Staubli VAL3: io.pjx

--- io.pjx ---
Parameters version=s7.2 stackSize=0 millimeterUnit=true
Data file=io.dtx

--- io.dtx ---
public aio CBT_TEMP = {link=CBT_TEMP}
public aio CPU_TEMP = {link=CPU_TEMP}
public aio MbAI_a8Axispose = {link=MbAI_a8Axispose}
public aio MbAI_aCurPosH = {link=MbAI_aCurPosH}
public aio MbAI_aCurPosL = {link=MbAI_aCurPosL}
public aio MbAI_aUnused4 = {link=MbAI_aUnused4}
public aio MbAI_b8MotorErr = {link=MbAI_b8MotorErr}
public aio MbAI_b8MotorPow = {link=MbAI_b8MotorPow}
public aio MbAI_bAxis7Reac = {link=MbAI_bAxis7Reac}
public aio MbAI_bAxis8Reac = {link=MbAI_bAxis8Reac}
public aio MbAI_bBackHome = {link=MbAI_bBackHome}
public aio MbAI_bDownLimit = {link=MbAI_bDownLimit}
public aio MbAI_bEndCycl = {link=MbAI_bEndCycl}
public aio MbAI_bHomeDone = {link=MbAI_bHomeDone}
public aio MbAI_bHomeLimit = {link=MbAI_bHomeLimit}
public aio MbAI_bIsHome = {link=MbAI_bIsHome}
public aio MbAI_bMotorErro = {link=MbAI_bMotorErro}
public aio MbAI_bMotorPowe = {link=MbAI_bMotorPowe}
public aio MbAI_bOutAlarm = {link=MbAI_bOutAlarm}
public aio MbAI_bPowerOn = {link=MbAI_bPowerOn}
public aio MbAI_bStartCycl = {link=MbAI_bStartCycl}
public aio MbAI_bUnused1 = {link=MbAI_bUnused1}
public aio MbAI_bUnused10 = {link=MbAI_bUnused10}
public aio MbAI_bUnused11 = {link=MbAI_bUnused11}
public aio MbAI_bUnused2 = {link=MbAI_bUnused2}
public aio MbAI_bUnused3 = {link=MbAI_bUnused3}
public aio MbAI_bUnused5 = {link=MbAI_bUnused5}
public aio MbAI_bUnused6 = {link=MbAI_bUnused6}
public aio MbAI_bUnused7 = {link=MbAI_bUnused7}
public aio MbAI_bUnused8 = {link=MbAI_bUnused8}
public aio MbAI_bUnused9 = {link=MbAI_bUnused9}
public aio MbAI_bUpLimit = {link=MbAI_bUpLimit}
public aio MbAO_aAxis7Puls = {link=MbAO_aAxis7Puls}
public aio MbAO_aAxis8Puls = {link=MbAO_aAxis8Puls}
public aio MbAO_aJogVelo = {link=MbAO_aJogVelo}
public aio MbAO_aJogVelo8 = {link=MbAO_aJogVelo8}
public aio MbAO_aMoveDis = {link=MbAO_aMoveDis}
public aio MbAO_aMoveDis8 = {link=MbAO_aMoveDis8}
public aio MbAO_aMovePosH = {link=MbAO_aMovePosH}
public aio MbAO_aMovePosH8 = {link=MbAO_aMovePosH8}
public aio MbAO_aMovePosL = {link=MbAO_aMovePosL}
public aio MbAO_aMovePosL8 = {link=MbAO_aMovePosL8}
public aio MbAO_aUnused10 = {link=MbAO_aUnused10}
public aio MbAO_aUnused11 = {link=MbAO_aUnused11}
public aio MbAO_aUnused6 = {link=MbAO_aUnused6}
public aio MbAO_aUnused7 = {link=MbAO_aUnused7}
public aio MbAO_aUnused8 = {link=MbAO_aUnused8}
public aio MbAO_aUnused9 = {link=MbAO_aUnused9}
public aio MbAO_aVelocity = {link=MbAO_aVelocity}
public aio MbAO_aVelocity8 = {link=MbAO_aVelocity8}
public aio MbAO_b7Axis = {link=MbAO_b7Axis}
public aio MbAO_b8Axis = {link=MbAO_b8Axis}
public aio MbAO_bAxis7Dire = {link=MbAO_bAxis7Dire}
public aio MbAO_bAxis7Home = {link=MbAO_bAxis7Home}
public aio MbAO_bAxis8Dire = {link=MbAO_bAxis8Dire}
public aio MbAO_bMoveDir = {link=MbAO_bMoveDir}
public aio MbAO_bMoveDirM = {link=MbAO_bMoveDirM}
public aio MbAO_bMovePos8 = {link=MbAO_bMovePos8}
public aio MbAO_bMoveToPos = {link=MbAO_bMoveToPos}
public aio MbAO_bRecordPos = {link=MbAO_bRecordPos}
public aio MbAO_bResetErr = {link=MbAO_bResetErr}
public aio MbAO_bStopMotor = {link=MbAO_bStopMotor}
public aio MbAO_bUnused1 = {link=MbAO_bUnused1}
public aio MbAO_bUnused2 = {link=MbAO_bUnused2}
public aio MbAO_bUnused3 = {link=MbAO_bUnused3}
public aio MbAO_bUnused4 = {link=MbAO_bUnused4}
public aio MbAO_bUnused5 = {link=MbAO_bUnused5}
public aio cCounts = {link=cCounts}
public aio cCurrPos = {link=cCurrPos}
public aio cLatchPos = {link=cLatchPos}
public aio cPrstPos = {link=cPrstPos}
public dio CASTING = {link=CASTING}
public dio DSI_BOARD = {link=DSI_BOARD}
public dio GLOBAL_PTC = {link=GLOBAL_PTC}
public dio MOTOR_1_3_5 = {link=MOTOR_1_3_5}
public dio MOTOR_2_4_6 = {link=MOTOR_2_4_6}
public dio SECTEUR_OK = {link=SECTEUR_OK}
public dio b2In0 = {link=BasicIO-2\%I0}
public dio b2In1 = {link=BasicIO-2\%I1}
public dio b2In10 = {link=BasicIO-2\%I10}
public dio b2In11 = {link=BasicIO-2\%I11}
public dio b2In12 = {link=BasicIO-2\%I12}
public dio b2In13 = {link=BasicIO-2\%I13}
public dio b2In14 = {link=BasicIO-2\%I14}
public dio b2In15 = {link=BasicIO-2\%I15}
public dio b2In2 = {link=BasicIO-2\%I2}
public dio b2In3 = {link=BasicIO-2\%I3}
public dio b2In4 = {link=BasicIO-2\%I4}
public dio b2In5 = {link=BasicIO-2\%I5}
public dio b2In6 = {link=BasicIO-2\%I6}
public dio b2In7 = {link=BasicIO-2\%I7}
public dio b2In8 = {link=BasicIO-2\%I8}
public dio b2In9 = {link=BasicIO-2\%I9}
public dio b2Out0 = {link=BasicIO-2\%Q0}
public dio b2Out1 = {link=BasicIO-2\%Q1}
public dio b2Out10 = {link=BasicIO-2\%Q10}
public dio b2Out11 = {link=BasicIO-2\%Q11}
public dio b2Out12 = {link=BasicIO-2\%Q12}
public dio b2Out13 = {link=BasicIO-2\%Q13}
public dio b2Out14 = {link=BasicIO-2\%Q14}
public dio b2Out15 = {link=BasicIO-2\%Q15}
public dio b2Out2 = {link=BasicIO-2\%Q2}
public dio b2Out3 = {link=BasicIO-2\%Q3}
public dio b2Out4 = {link=BasicIO-2\%Q4}
public dio b2Out5 = {link=BasicIO-2\%Q5}
public dio b2Out6 = {link=BasicIO-2\%Q6}
public dio b2Out7 = {link=BasicIO-2\%Q7}
public dio b2Out8 = {link=BasicIO-2\%Q8}
public dio b2Out9 = {link=BasicIO-2\%Q9}
public dio bIn0 = {link=BasicIO-1\%I0}
public dio bIn1 = {link=BasicIO-1\%I1}
public dio bIn10 = {link=BasicIO-1\%I10}
public dio bIn11 = {link=BasicIO-1\%I11}
public dio bIn12 = {link=BasicIO-1\%I12}
public dio bIn13 = {link=BasicIO-1\%I13}
public dio bIn14 = {link=BasicIO-1\%I14}
public dio bIn15 = {link=BasicIO-1\%I15}
public dio bIn2 = {link=BasicIO-1\%I2}
public dio bIn3 = {link=BasicIO-1\%I3}
public dio bIn4 = {link=BasicIO-1\%I4}
public dio bIn5 = {link=BasicIO-1\%I5}
public dio bIn6 = {link=BasicIO-1\%I6}
public dio bIn7 = {link=BasicIO-1\%I7}
public dio bIn8 = {link=BasicIO-1\%I8}
public dio bIn9 = {link=BasicIO-1\%I9}
public dio bOut0 = {link=BasicIO-1\%Q0}
public dio bOut1 = {link=BasicIO-1\%Q1}
public dio bOut10 = {link=BasicIO-1\%Q10}
public dio bOut11 = {link=BasicIO-1\%Q11}
public dio bOut12 = {link=BasicIO-1\%Q12}
public dio bOut13 = {link=BasicIO-1\%Q13}
public dio bOut14 = {link=BasicIO-1\%Q14}
public dio bOut15 = {link=BasicIO-1\%Q15}
public dio bOut2 = {link=BasicIO-1\%Q2}
public dio bOut3 = {link=BasicIO-1\%Q3}
public dio bOut4 = {link=BasicIO-1\%Q4}
public dio bOut5 = {link=BasicIO-1\%Q5}
public dio bOut6 = {link=BasicIO-1\%Q6}
public dio bOut7 = {link=BasicIO-1\%Q7}
public dio bOut8 = {link=BasicIO-1\%Q8}
public dio bOut9 = {link=BasicIO-1\%Q9}
public dio cEnLatch = {link=cEnLatch}
public dio cEnPrst = {link=cEnPrst}
public dio cHwErr = {link=cHwErr}
public dio cLatch = {link=cLatch}
public dio cOvsErr = {link=cOvsErr}
public dio cRstErr = {link=cRstErr}
public dio fIn0 = {link=fIn0}
public dio fIn1 = {link=fIn1}
public dio fOut0 = {link=fOut0}
public dio usrIn0 = {link=usrIn0}
public dio usrIn1 = {link=usrIn1}
public dio valve1 = {link=valve1}
public dio valve2 = {link=valve2}
public sio socket = {link=socket}
